// TIA Portal V17 export
// export: Created 2025-05-22T06:00:42.1709528Z, ExportSetting WithDefaults, DisplayName Totally Integrated Automation Portal, DisplayVersion V17 Update 8, DisplayName TIA Portal Openness, DisplayVersion V17 Update 8, DisplayName TIA Portal Version Control Interface, DisplayVersion V17, DisplayName SINAMICS Startdrive Advanced, DisplayVersion V17 SP2, DisplayName SINAMICS Startdrive G110M, G120, G120C, G120D, G120P, G115D, DisplayVersion V17 SP2, DisplayName SINAMICS Startdrive G130, G150, S120, S150, SINAMICS MV, S210, DisplayVersion V17 SP2, DisplayName STEP 7 Professional, DisplayVersion V17 Update 8, DisplayName SINUMERIK ONE STEP 7 Toolbox, DisplayVersion V17 Update 12, DisplayName SINUMERIK ONE PLC Basic Program Plus, DisplayVersion V17 Update 12, DisplayName SINUMERIK 840D sl STEP 7 Toolbox, DisplayVersion V17 Update 12, DisplayName STEP 7 Safety, DisplayVersion V17 Update 6, DisplayName WinCC Advanced, DisplayVersion V17 Update 8
FUNCTION "FC7202_MESSAGES" : Void   // FC7202, LAD
TITLE = GRUPOS DATOS DIFERENTES A CERO
{ S7_Optimized_Access := 'FALSE' }
AUTHOR : ETXETAR
VERSION : 1.0
// Gestiona si el grupo de datos son diferentes a cero
// DB1980.DBX0.0 debe ser =0
// DB1980.DBX0.1 debe ser =1
// stored: AutoNumber false, IsIECCheckEnabled false, SetENOAutomatically false, UDAEnableTagReadback false
   VAR_INPUT
      DB : DB_ANY;
      "BEGIN" : Int;
      BYTES : Int;
   END_VAR
   VAR_OUTPUT
      OUTPUT : Bool;
   END_VAR
   VAR_TEMP
      AUX_1 : Word;
      AUX_2 : Word;
      AUX_OUT_1 : Bool;
   END_VAR
BEGIN

NETWORK
TITLE = 
// Grupo de datos:
      A     "M_ZERO";
      =     #OUTPUT;  // INITIALIZE OUTPUT
      L     0;
      T     #AUX_1;  // INITIALIZE LOCAL VARIABLES
      T     #AUX_2;
      L     P#0.0;  // INITIALIZE POINTER
      LAR1;

      OPN   #DB;  // OPEN DB
      L     #"BEGIN";
      T     #AUX_1;
      L     #BYTES;
M002: T     #AUX_2;
      L     #AUX_1;
      SLW   3;
      LAR1;

      OPN   #DB;
      L     DBB [AR1, P#0.0];
      L     0;
      ==I;
      JC    M005;
      JU    M001;
M005: L     #AUX_1;
      L     1;
      +I;
      T     #AUX_1;
      L     #AUX_2;
      LOOP  M002;
      A     "M_ZERO";
      =     #AUX_OUT_1;
      JU    M003;
M001: A     "M_ONE";
      =     #AUX_OUT_1;
M003: NOP   0;


REGION Network 2
   // Activa la salida
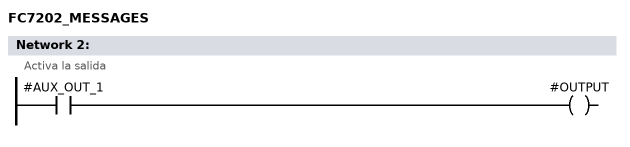
   RUNG wire#powerrail
      Contact( #AUX_OUT_1 )
      Coil( #OUTPUT )
   END_RUNG
   // the same network as SCL:
   #OUTPUT := #AUX_OUT_1;
END_REGION
END_FUNCTION
